{attribute addProperty BoxType "EL2262-0000-0002"}
{attribute addProperty Id "CycCount0AT %Q*CycCount0_307034DC1620Sample0AT %Q*ARRAY[0..9] OF Sample_ABF5BEA980100GapAT %Q*EMPTY_STRUCTURE000CycCount1AT %Q*CycCount1_7787FA1D1620Sample1AT %Q*ARRAY[0..9] OF Sample_4351E8AC80100Gap_1AT %Q*EMPTY_STRUCTURE000WcStateAT %I*WcState_64F6A8C6810InfoDataAT %I*InfoData_7231B2DD80100"}
{attribute addProperty CRC "3930548172"}
{attribute addProperty SizeInBites "280"}
{attribute addProperty SizeInBytes "35"}
TYPE EL2262_A80E6C9A :
STRUCT
	{attribute addProperty Name "CycCount0"}
	CycCount0 : CycCount0_307034DC;
	{attribute addProperty Name "Sample0"}
	Sample0 : ARRAY[0..9] OF Sample_ABF5BEA9;
	{attribute addProperty Name "Gap"}
	Gap : EMPTY_STRUCTURE;
	{attribute addProperty Name "CycCount1"}
	CycCount1 : CycCount1_7787FA1D;
	{attribute addProperty Name "Sample1"}
	Sample1 : ARRAY[0..9] OF Sample_4351E8AC;
	{attribute addProperty Name "Gap_1"}
	Gap_1 : EMPTY_STRUCTURE;
	{attribute addProperty Name "WcState"}
	WcState : WcState_64F6A8C6;
	{attribute addProperty Name "InfoData"}
	InfoData : InfoData_7231B2DD;
END_STRUCT
END_TYPE

(* stored: Version 1.2.0.0, ProductVersion 3.1.4024.9
   DUT EL2262_A80E6C9A: Id {6650e348-a634-4658-9026-abd0b736d8f5} *)
